// TIA Portal V20 export
TYPE "TypeDOL"
// stored: IsFailsafeCompliant false
   STRUCT
      Run : Bool;
      FaultActive : Bool;
      SpeedSetpoint : Real;
      RunHours : UDInt;
      StatusWord : Word;
      EquipmentName : String;
   END_STRUCT;
END_TYPE
